# EPICS autosave request: ttiMX/ttiMX_channel_settings.req
$(P):$(CHAN):CURRENT
$(P):$(CHAN):OUTPUT
$(P):$(CHAN):VOLTAGE
$(P):$(CHAN):VRANGE
